# EPICS autosave request: iocBoot/ioc13xps_test/auto_settings.req
file "CARS_motor_settings.req",         P=13xps3:, M=m1
